FUNCTION_BLOCK TINA_0
  {SET_ATTRIBUTE(OpcUa, DEVICE.EQUIPMENT)}
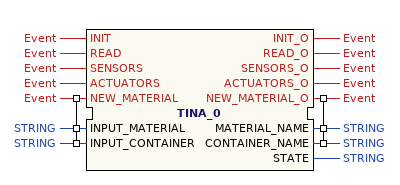
  EVENT_INPUT
    INIT;
    READ;
    SENSORS;
    ACTUATORS;
    NEW_MATERIAL WITH INPUT_MATERIAL, INPUT_CONTAINER;
  END_EVENT
  EVENT_OUTPUT
    INIT_O;
    READ_O;
    SENSORS_O;
    ACTUATORS_O;
    NEW_MATERIAL_O WITH MATERIAL_NAME, CONTAINER_NAME;
  END_EVENT
  VAR_INPUT
    INPUT_MATERIAL : STRING; {SET_ATTRIBUTE(OpcUa, Variable)}
    INPUT_CONTAINER : STRING; {SET_ATTRIBUTE(OpcUa, Variable)}
  END_VAR
  VAR_OUTPUT
    MATERIAL_NAME : STRING; {SET_ATTRIBUTE(OpcUa, Variable)}
    CONTAINER_NAME : STRING; {SET_ATTRIBUTE(OpcUa, Variable)}
    STATE : STRING; {SET_ATTRIBUTE(OpcUa, Variable)}
  END_VAR
END_FUNCTION_BLOCK
